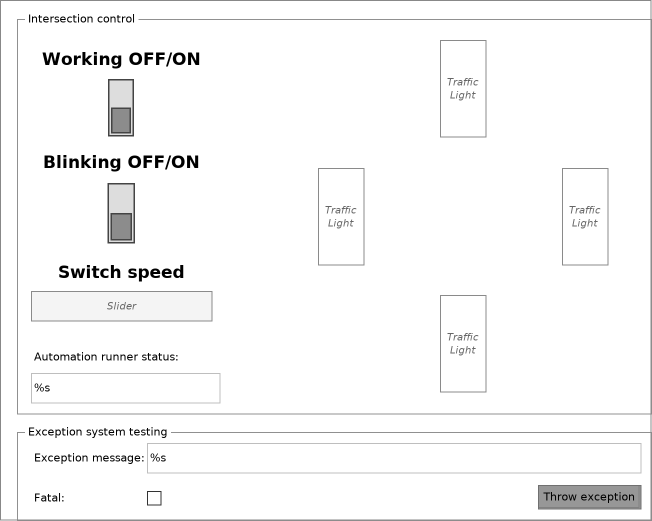
VISUALIZATION MainWindow  // 652x521
    GroupBox (17,11 635x403), "Intersection control"
        Rectangle (385,25 120x360), angle 90
        Label (17,33 175x30), "Working OFF/ON"
        Label (17,136 175x30), "Blinking OFF/ON"
        Line (328,119)
        Rectangle (385,17 120x376)
        Frame (423,29 46x97)
            shows TrafficLight(Red := MAIN.AutomationRunner.SignalControlledIntersectionAutomationController.TrafficLight2.RedLight.SimulatedContactValue, Yellow := MAIN.AutomationRunner.SignalControlledIntersectionAutomationController.TrafficLight2.YellowLight.SimulatedContactValue, Green := MAIN.AutomationRunner.SignalControlledIntersectionAutomationController.TrafficLight2.GreenLight.SimulatedContactValue)
        Frame (423,284 46x97)
            shows TrafficLight(Red := MAIN.AutomationRunner.SignalControlledIntersectionAutomationController.TrafficLight4.RedLight.SimulatedContactValue, Yellow := MAIN.AutomationRunner.SignalControlledIntersectionAutomationController.TrafficLight4.YellowLight.SimulatedContactValue, Green := MAIN.AutomationRunner.SignalControlledIntersectionAutomationController.TrafficLight4.GreenLight.SimulatedContactValue)
        Frame (545,157 46x97)
            shows TrafficLight(Red := MAIN.AutomationRunner.SignalControlledIntersectionAutomationController.TrafficLight3.RedLight.SimulatedContactValue, Yellow := MAIN.AutomationRunner.SignalControlledIntersectionAutomationController.TrafficLight3.YellowLight.SimulatedContactValue, Green := MAIN.AutomationRunner.SignalControlledIntersectionAutomationController.TrafficLight3.GreenLight.SimulatedContactValue)
        Frame (301,157 46x97)
            shows TrafficLight(Red := MAIN.AutomationRunner.SignalControlledIntersectionAutomationController.TrafficLight1.RedLight.SimulatedContactValue, Yellow := MAIN.AutomationRunner.SignalControlledIntersectionAutomationController.TrafficLight1.YellowLight.SimulatedContactValue, Green := MAIN.AutomationRunner.SignalControlledIntersectionAutomationController.TrafficLight1.GreenLight.SimulatedContactValue)
        DipSwitch (64,68 80x57), variable: MAIN.AutomationRunner.SignalControlledIntersectionAutomationController.WorkingModeSwitch.SimulatedContactValue, behaviour: TOGGLE, style: Switch-DipSwitch-Gray
        DipSwitch (64,172 80x60), variable: MAIN.AutomationRunner.SignalControlledIntersectionAutomationController.BlinkingYellowModeSwitch.SimulatedContactValue, behaviour: TOGGLE, style: Switch-DipSwitch-Gray
        Textfield (14,362 189x30), "%s", text variable: MAIN.AutomationRunner.StateName, input disabled if: FALSE
        Label (14,331 150x30), "Automation runner status:"
        Slider (14,280 181x30), variable: MAIN.AutomationRunner.SignalControlledIntersectionAutomationController.SwitchSpeedAdjuster.SimulatedDigitizedValue._16Bit, scale -32768..32767
        Label (17,246 175x30), "Switch speed"
    GroupBox (17,424 635x97), "Exception system testing"
        Label (14,19 116x30), "Exception message:"
        Textfield (130,19 494x30), "%s", text variable: MAIN.AutomationRunner.SignalControlledIntersectionAutomationController.TestExceptionMessage, input disabled if: FALSE
            OnMouseClick: write the text variable via Default
        Button (521,61 103x24), "Throw exception"
            OnMouseClick: execute { MAIN.AutomationRunner.SignalControlledIntersectionAutomationController.ThrowTestExceptionRequest := TRUE; }
        Checkbox (128,59 34x30), variable: MAIN.AutomationRunner.SignalControlledIntersectionAutomationController.IsTestExceptionFatal
        Label (14,59 110x30), "Fatal:"
END_VISUALIZATION

(* stored: Version 1.1.0.1
   Visu MainWindow: Id {3f36056b-e97d-47c4-837d-733890435638} *)
